TYPE stAxisIF :
STRUCT
END_STRUCT
END_TYPE

(* stored: Version 1.1.0.1, ProductVersion 3.1.4024.3
   DUT stAxisIF: Id {ccfbe191-241f-0f82-1c8c-4ecf1fcd274b} *)
